PROGRAM MAIN
VAR
	Q01 : BOOL;
	S01 : BOOL;
END_VAR

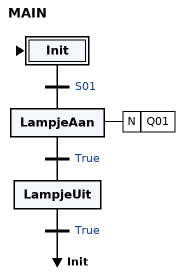
INITIAL_STEP Init:
END_STEP
TRANSITION FROM Init TO LampjeAan
    := S01;
END_TRANSITION
STEP LampjeAan:  // min time t#700ms
    Q01(N);
END_STEP
TRANSITION FROM LampjeAan TO LampjeUit
    := True;
END_TRANSITION
STEP LampjeUit:  // min time t#300ms
END_STEP
TRANSITION FROM LampjeUit TO Init
    := True;
END_TRANSITION

END_PROGRAM

(* stored: Version 1.1.0.1, ProductVersion 3.1.4024.12
   POU MAIN: Id {ea707d9c-b6f3-44e8-8dec-e576531839b3}, SpecialFunc None *)
